(* Schneider Machine Expert - Basic project Prototype 1 Mod, file version 2.7.0.0 *)
(* ProjectInformations: Name=Nuevo proyecto *)

HARDWARE
  Cpu 0: TM221M16R/G
  ModuleExtensionObject 0: TM3DI16K
  ModuleExtensionObject 1: TM3AQ2/G
  ModuleExtensionObject 2: TM3AQ4/G
  ModuleExtensionObject 3: TM3DQ16R/G
  EthernetConfiguration: NetworkName=M221, IpAllocationMode=FixedAddress, IpAddress=0.0.0.0, SubnetMask=0.0.0.0
  SerialLineConfiguration: Baud=Baud19200, Parity=ParityEven, DataBits=DataBits8, StopBits=StopBits1, PhysicalMedium=PhysicalMediumRs485, TransmissionMode=TransmissionModeModbusRtu, SlaveId=1, Addressing=SlaveAddressing
  MastTask: UsePeriodScanMode=false, PeriodScan=100
  FastTask: Period=255
  CpuBehavior: StartingMode=StartAsPreviousState, AutoSaveRamOnEeprom=true, WatchdogPeriod=250

SYMBOLS  (address, symbol, comment, settings)
  %M0       START_BUTTON
  %M1       RESET_BUTTON
  %M2       STOP_BUTTON
  %M3       EMERGENCY_BUTTON
  %M4       AUTO_SWITCH
  %M5       ENTRY_SENSOR
  %M7       PERSON
  %M8       EXIT_SENSOR
  %M9       COUNTER_SENSOR
  %M10      ITEM_DETECTED_1
  %M11      ITEM_DETECTED_2
  %M13      MOVING_XY_1
  %M16      MOVING_Z1
  %M18      ENTRY_CONVEYOR
  %M19      MIDDLE_CONVEYOR
  %M20      EXIT_CONVEYOR
  %M21      GRAB_1
  %M22      GRAB_2
  %M23      START_LIGHT
  %M24      RESET_LIGHT
  %M25      STOP_LIGHT
  %M26      RED_LIGHT
  %M27      YELLOW_LIGHT
  %M28      GREEN_LIGHT
  %M29      ALARM
  %M100     INITIALIZE
  %M101     INITIAL_POS_1
  %M102     INITIAL_POS_2
  %M200     FLAG_AUTO
  %S21      SB_INITGRAFCET  "En el estado 1, este bit provoca una inicialización GRAFCET. Los pasos activos se desactivan y los pasos iniciales se activan"
  %X1       STATE_1
  %X2       STATE_2
  %X3       STATE_3
  %X4       STATE_4
  %X5       STATE_5
  %X6       STATE_6
  %X7       STATE_7
  %X8       STATE_8
  %X9       STATE_9
  %X10      STATE_10
  %X11      STATE_11
  %X12      STATE_12
  %X13      STATE_13
  %X14      STATE_14
  %X15      STATE_15
  %X16      STATE_16
  %X17      STATE_17
  %X18      STATE_18
  %X19      STATE_19
  %X21      STATE_21
  %MW0      X1
  %MW1      Y1
  %MW2      Z1
  %MW3      X2
  %MW4      Y2
  %MW5      Z2
  %MW6      X1_MOVE
  %MW7      Y1_MOVE
  %MW8      Z1_MOVE
  %MW9      X2_MOVE
  %MW10     Y2_MOVE
  %MW11     Z2_MOVE
  %MW12     COUNTER_OF_ITEMS
  %TM0      TIME_OF_OPERATION  [Preset=10, Base=OneSecond]
  %TM1      SECURITY_TIME  [Preset=5, Base=OneSecond]
  %TM2        "Syren time"  [Type=TOF, Preset=30, Base=OneSecond]
  %C0       NUMBER_OF_ITEMS

GRAFCET Grafcet
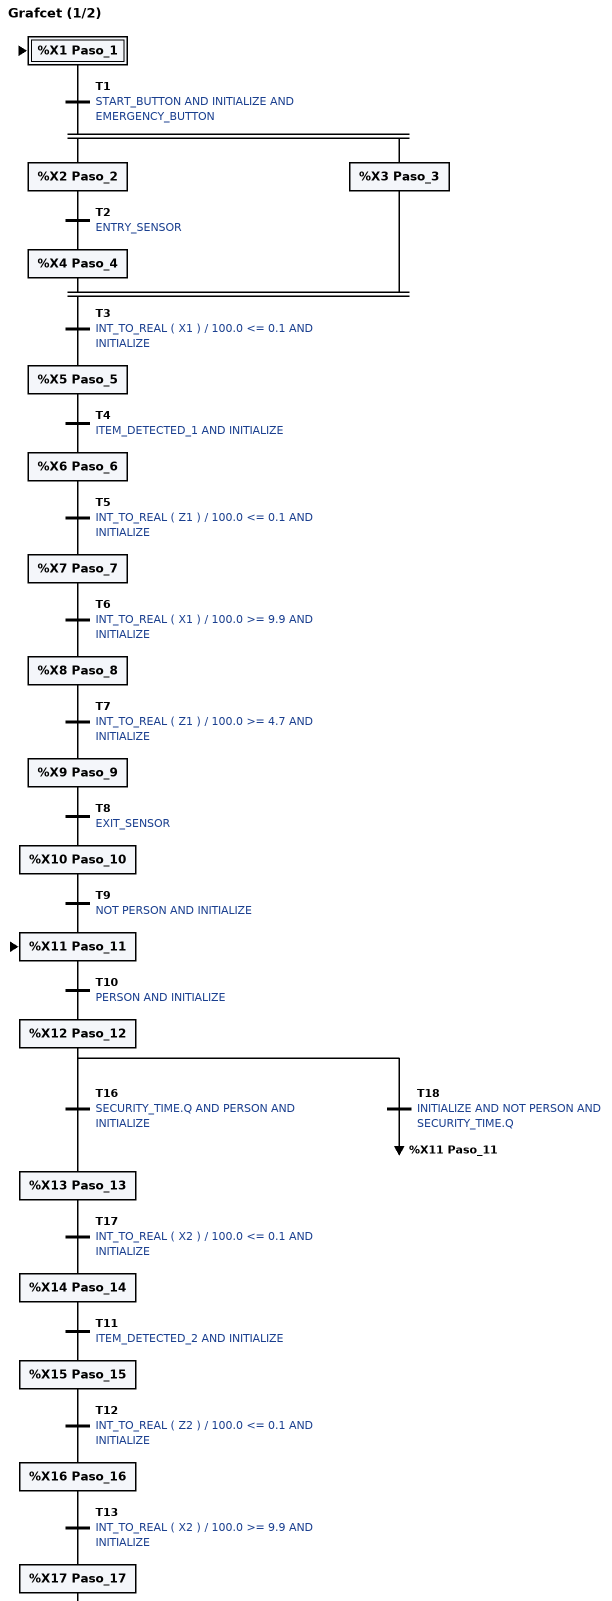
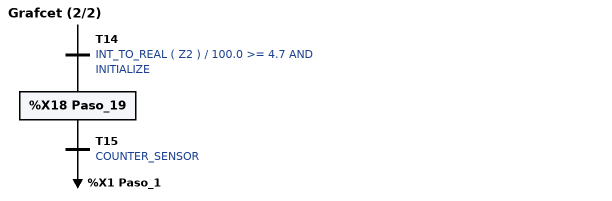
  INITIAL_STEP %X1  (* Paso_1 *)
  STEP %X2  (* Paso_2 *)
  STEP %X3  (* Paso_3 *)
  STEP %X4  (* Paso_4 *)
  STEP %X5  (* Paso_5 *)
  STEP %X6  (* Paso_6 *)
  STEP %X7  (* Paso_7 *)
  STEP %X8  (* Paso_8 *)
  STEP %X9  (* Paso_9 *)
  STEP %X10  (* Paso_10 *)
  STEP %X11  (* Paso_11 *)
  STEP %X12  (* Paso_12 *)
  STEP %X13  (* Paso_13 *)
  STEP %X14  (* Paso_14 *)
  STEP %X15  (* Paso_15 *)
  STEP %X16  (* Paso_16 *)
  STEP %X17  (* Paso_17 *)
  STEP %X18  (* Paso_19 *)
  TRANSITION T1 FROM %X1 TO %X2, %X3 := START_BUTTON AND INITIALIZE AND EMERGENCY_BUTTON;
  TRANSITION T2 FROM %X2 TO %X4 := ENTRY_SENSOR;
  TRANSITION T3 FROM %X4, %X3 TO %X5 := INT_TO_REAL ( X1 ) / 100.0 <= 0.1 AND INITIALIZE;
  TRANSITION T4 FROM %X5 TO %X6 := ITEM_DETECTED_1 AND INITIALIZE;
  TRANSITION T5 FROM %X6 TO %X7 := INT_TO_REAL ( Z1 ) / 100.0 <= 0.1 AND INITIALIZE;
  TRANSITION T6 FROM %X7 TO %X8 := INT_TO_REAL ( X1 ) / 100.0 >= 9.9 AND INITIALIZE;
  TRANSITION T7 FROM %X8 TO %X9 := INT_TO_REAL ( Z1 ) / 100.0 >= 4.7 AND INITIALIZE;
  TRANSITION T8 FROM %X9 TO %X10 := EXIT_SENSOR;
  TRANSITION T9 FROM %X10 TO %X11 := NOT PERSON AND INITIALIZE;
  TRANSITION T10 FROM %X11 TO %X12 := PERSON AND INITIALIZE;
  TRANSITION T11 FROM %X14 TO %X15 := ITEM_DETECTED_2 AND INITIALIZE;
  TRANSITION T12 FROM %X15 TO %X16 := INT_TO_REAL ( Z2 ) / 100.0 <= 0.1 AND INITIALIZE;
  TRANSITION T13 FROM %X16 TO %X17 := INT_TO_REAL ( X2 ) / 100.0 >= 9.9 AND INITIALIZE;
  TRANSITION T14 FROM %X17 TO %X18 := INT_TO_REAL ( Z2 ) / 100.0 >= 4.7 AND INITIALIZE;
  TRANSITION T15 FROM %X18 TO %X1 := COUNTER_SENSOR;
  TRANSITION T16 FROM %X12 TO %X13 := SECURITY_TIME.Q AND PERSON AND INITIALIZE;
  TRANSITION T17 FROM %X13 TO %X14 := INT_TO_REAL ( X2 ) / 100.0 <= 0.1 AND INITIALIZE;
  TRANSITION T18 FROM %X12 TO %X11 := INITIALIZE AND NOT PERSON AND SECURITY_TIME.Q;

TRANSITION T1 (%X1 -> %X2, %X3) 
  (* SectionNumber=0 *)

// Rung 0: Tr1
  LD %M0                  (* START_BUTTON *)
  AND %M100               (* INITIALIZE *)
  AND %M3                 (* EMERGENCY_BUTTON *)
  ENDT
  // as ST:
  //   TRANSITION := START_BUTTON AND INITIALIZE AND EMERGENCY_BUTTON;

TRANSITION T2 (%X2 -> %X4) 
  (* SectionNumber=0 *)

// Rung 1: Tr2
  LD %M5                  (* ENTRY_SENSOR *)
  ENDT
  // as ST:
  //   TRANSITION := ENTRY_SENSOR;

TRANSITION T3 (%X4, %X3 -> %X5) 
  (* SectionNumber=0 *)

// Rung 2: Tr3
  LD 1
  AND [ INT_TO_REAL ( %MW0 ) / 100.0 <= 0.1 ](* X1 *)
  AND %M100               (* INITIALIZE *)
  ENDT
  // as ST:
  //   TRANSITION := INT_TO_REAL ( X1 ) / 100.0 <= 0.1 AND INITIALIZE;

TRANSITION T4 (%X5 -> %X6) 
  (* SectionNumber=0 *)

// Rung 3: Tr4
  LD %M10                 (* ITEM_DETECTED_1 *)
  AND %M100               (* INITIALIZE *)
  ENDT
  // as ST:
  //   TRANSITION := ITEM_DETECTED_1 AND INITIALIZE;

TRANSITION T5 (%X6 -> %X7) 
  (* SectionNumber=0 *)

// Rung 4: Tr5
  LD 1
  AND [ INT_TO_REAL ( %MW2 ) / 100.0 <= 0.1 ](* Z1 *)
  AND %M100               (* INITIALIZE *)
  ENDT
  // as ST:
  //   TRANSITION := INT_TO_REAL ( Z1 ) / 100.0 <= 0.1 AND INITIALIZE;

TRANSITION T6 (%X7 -> %X8) 
  (* SectionNumber=0 *)

// Rung 5: Tr6
  LD 1
  AND [ INT_TO_REAL ( %MW0 ) / 100.0 >= 9.9 ](* X1 *)
  AND %M100               (* INITIALIZE *)
  ENDT
  // as ST:
  //   TRANSITION := INT_TO_REAL ( X1 ) / 100.0 >= 9.9 AND INITIALIZE;

TRANSITION T7 (%X8 -> %X9) 
  (* SectionNumber=0 *)

// Rung 6: Tr7
  LD 1
  AND [ INT_TO_REAL ( %MW2 ) / 100.0 >= 4.7 ](* Z1 *)
  AND %M100               (* INITIALIZE *)
  ENDT
  // as ST:
  //   TRANSITION := INT_TO_REAL ( Z1 ) / 100.0 >= 4.7 AND INITIALIZE;

TRANSITION T8 (%X9 -> %X10) 
  (* SectionNumber=0 *)

// Rung 7: Tr8
  LD %M8                  (* EXIT_SENSOR *)
  ENDT
  // as ST:
  //   TRANSITION := EXIT_SENSOR;

TRANSITION T9 (%X10 -> %X11) 
  (* SectionNumber=0 *)

// Rung 8: Tr9
  LDN %M7                 (* PERSON *)
  AND %M100               (* INITIALIZE *)
  ENDT
  // as ST:
  //   TRANSITION := NOT PERSON AND INITIALIZE;

TRANSITION T10 (%X11 -> %X12) 
  (* SectionNumber=0 *)

// Rung 9: Tr10
  LD %M7                  (* PERSON *)
  AND %M100               (* INITIALIZE *)
  ENDT
  // as ST:
  //   TRANSITION := PERSON AND INITIALIZE;

TRANSITION T11 (%X14 -> %X15) 
  (* SectionNumber=0 *)

// Rung 10: Tr14
  LD %M11                 (* ITEM_DETECTED_2 *)
  AND %M100               (* INITIALIZE *)
  ENDT
  // as ST:
  //   TRANSITION := ITEM_DETECTED_2 AND INITIALIZE;

TRANSITION T12 (%X15 -> %X16) 
  (* SectionNumber=0 *)

// Rung 11: Tr15
  LD 1
  AND [ INT_TO_REAL ( %MW5 ) / 100.0 <= 0.1 ](* Z2 *)
  AND %M100               (* INITIALIZE *)
  ENDT
  // as ST:
  //   TRANSITION := INT_TO_REAL ( Z2 ) / 100.0 <= 0.1 AND INITIALIZE;

TRANSITION T13 (%X16 -> %X17) 
  (* SectionNumber=0 *)

// Rung 12: Tr16
  LD 1
  AND [ INT_TO_REAL ( %MW3 ) / 100.0 >= 9.9 ](* X2 *)
  AND %M100               (* INITIALIZE *)
  ENDT
  // as ST:
  //   TRANSITION := INT_TO_REAL ( X2 ) / 100.0 >= 9.9 AND INITIALIZE;

TRANSITION T14 (%X17 -> %X18) 
  (* SectionNumber=0 *)

// Rung 13: Tr17
  LD 1
  AND [ INT_TO_REAL ( %MW5 ) / 100.0 >= 4.7 ](* Z2 *)
  AND %M100               (* INITIALIZE *)
  ENDT
  // as ST:
  //   TRANSITION := INT_TO_REAL ( Z2 ) / 100.0 >= 4.7 AND INITIALIZE;

TRANSITION T15 (%X18 -> %X1) 
  (* SectionNumber=0 *)

// Rung 14: Tr18
  LD %M9                  (* COUNTER_SENSOR *)
  ENDT
  // as ST:
  //   TRANSITION := COUNTER_SENSOR;

TRANSITION T16 (%X12 -> %X13) 
  (* SectionNumber=0 *)

// Rung 15: Tr12
  LD %TM1.Q               (* SECURITY_TIME *)
  AND %M7                 (* PERSON *)
  AND %M100               (* INITIALIZE *)
  ENDT
  // as ST:
  //   TRANSITION := SECURITY_TIME.Q AND PERSON AND INITIALIZE;

TRANSITION T17 (%X13 -> %X14) 
  (* SectionNumber=0 *)

// Rung 16: Tr13
  LD 1
  AND [ INT_TO_REAL ( %MW3 ) / 100.0 <= 0.1 ](* X2 *)
  AND %M100               (* INITIALIZE *)
  ENDT
  // as ST:
  //   TRANSITION := INT_TO_REAL ( X2 ) / 100.0 <= 0.1 AND INITIALIZE;

TRANSITION T18 (%X12 -> %X11) 
  (* SectionNumber=0 *)

// Rung 17: Tr11
  LD %M100                (* INITIALIZE *)
  ANDN %M7                (* PERSON *)
  AND %TM1.Q              (* SECURITY_TIME *)
  ENDT
  // as ST:
  //   TRANSITION := INITIALIZE AND NOT PERSON AND SECURITY_TIME.Q;

POU Actions
  (* SectionNumber=20 *)

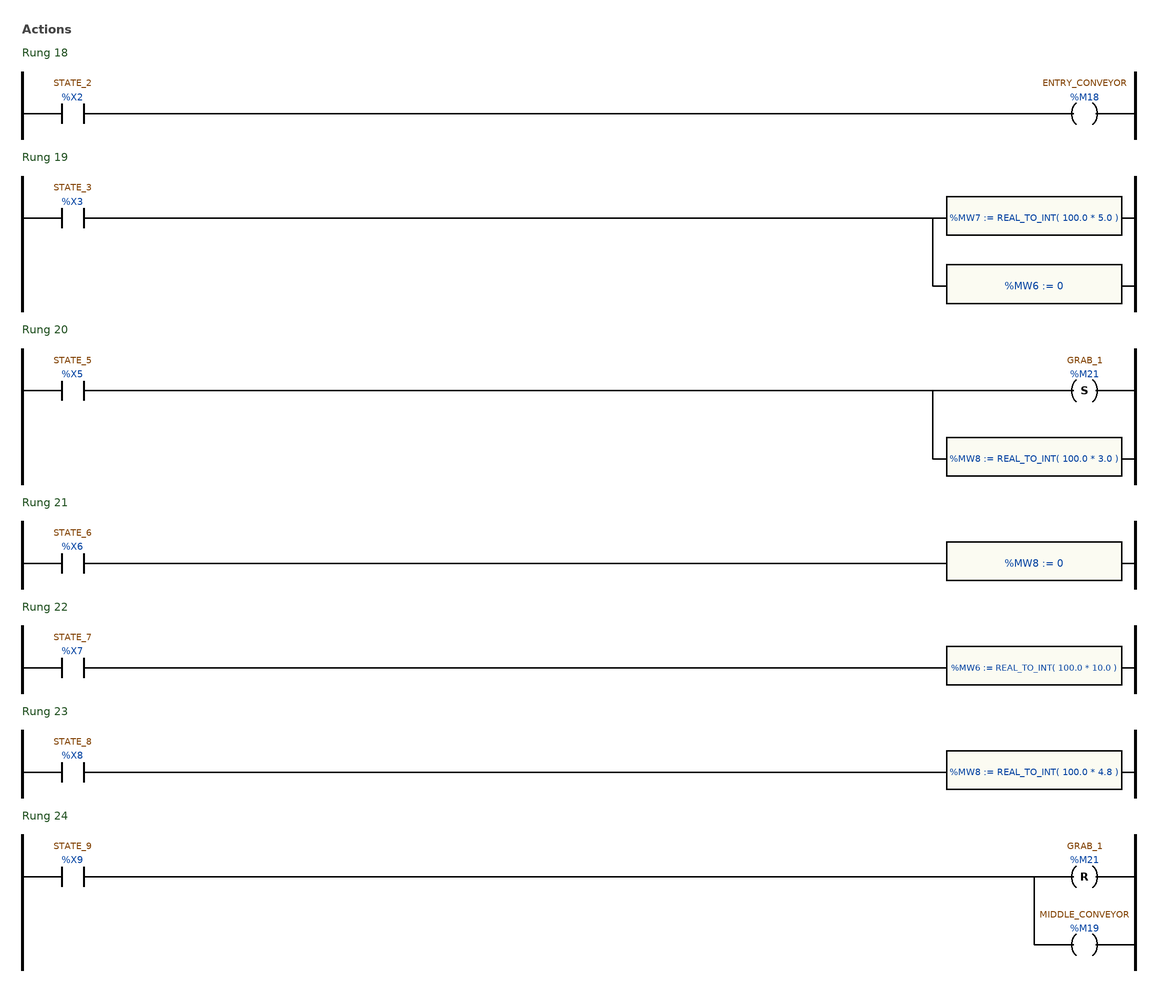

// Rung 18
  LD %X2                  (* STATE_2 *)
  ST %M18                 (* ENTRY_CONVEYOR *)
  // as ST:
  //   ENTRY_CONVEYOR := STATE_2;

// Rung 19
  LD %X3                  (* STATE_3 *)
  [ %MW7 := REAL_TO_INT ( 100.0 * 5.0 ) ](* Y1_MOVE *)
  [ %MW6 := 0 ]           (* X1_MOVE *)
  // as ST:
  //   IF STATE_3 THEN Y1_MOVE := REAL_TO_INT ( 100.0 * 5.0 ); END_IF;
  //   IF STATE_3 THEN X1_MOVE := 0; END_IF;

// Rung 20
  LD %X5                  (* STATE_5 *)
  S %M21                  (* GRAB_1 *)
  [ %MW8 := REAL_TO_INT ( 100.0 * 3.0 ) ](* Z1_MOVE *)
  // as ST:
  //   IF STATE_5 THEN GRAB_1 := TRUE; END_IF;
  //   IF STATE_5 THEN Z1_MOVE := REAL_TO_INT ( 100.0 * 3.0 ); END_IF;

// Rung 21
  LD %X6                  (* STATE_6 *)
  [ %MW8 := 0 ]           (* Z1_MOVE *)
  // as ST:
  //   IF STATE_6 THEN Z1_MOVE := 0; END_IF;

// Rung 22
  LD %X7                  (* STATE_7 *)
  [ %MW6 := REAL_TO_INT ( 100.0 * 10.0 ) ](* X1_MOVE *)
  // as ST:
  //   IF STATE_7 THEN X1_MOVE := REAL_TO_INT ( 100.0 * 10.0 ); END_IF;

// Rung 23
  LD %X8                  (* STATE_8 *)
  [ %MW8 := REAL_TO_INT ( 100.0 * 4.8 ) ](* Z1_MOVE *)
  // as ST:
  //   IF STATE_8 THEN Z1_MOVE := REAL_TO_INT ( 100.0 * 4.8 ); END_IF;

// Rung 24
  LD %X9                  (* STATE_9 *)
  R %M21                  (* GRAB_1 *)
  ST %M19                 (* MIDDLE_CONVEYOR *)
  // as ST:
  //   IF STATE_9 THEN GRAB_1 := FALSE; END_IF;
  //   MIDDLE_CONVEYOR := STATE_9;

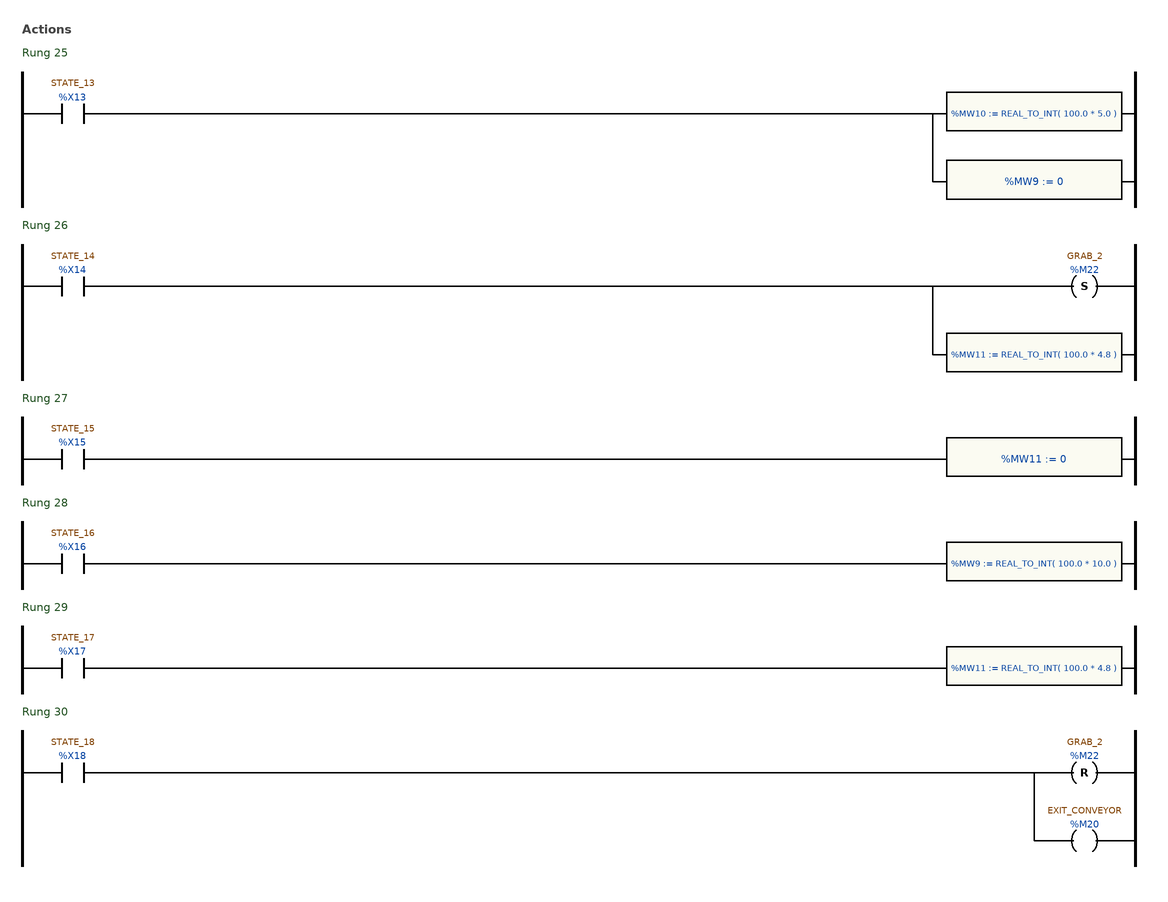

// Rung 25
  LD %X13                 (* STATE_13 *)
  [ %MW10 := REAL_TO_INT ( 100.0 * 5.0 ) ](* Y2_MOVE *)
  [ %MW9 := 0 ]           (* X2_MOVE *)
  // as ST:
  //   IF STATE_13 THEN Y2_MOVE := REAL_TO_INT ( 100.0 * 5.0 ); END_IF;
  //   IF STATE_13 THEN X2_MOVE := 0; END_IF;

// Rung 26
  LD %X14                 (* STATE_14 *)
  S %M22                  (* GRAB_2 *)
  [ %MW11 := REAL_TO_INT ( 100.0 * 4.8 ) ](* Z2_MOVE *)
  // as ST:
  //   IF STATE_14 THEN GRAB_2 := TRUE; END_IF;
  //   IF STATE_14 THEN Z2_MOVE := REAL_TO_INT ( 100.0 * 4.8 ); END_IF;

// Rung 27
  LD %X15                 (* STATE_15 *)
  [ %MW11 := 0 ]          (* Z2_MOVE *)
  // as ST:
  //   IF STATE_15 THEN Z2_MOVE := 0; END_IF;

// Rung 28
  LD %X16                 (* STATE_16 *)
  [ %MW9 := REAL_TO_INT ( 100.0 * 10.0 ) ](* X2_MOVE *)
  // as ST:
  //   IF STATE_16 THEN X2_MOVE := REAL_TO_INT ( 100.0 * 10.0 ); END_IF;

// Rung 29
  LD %X17                 (* STATE_17 *)
  [ %MW11 := REAL_TO_INT ( 100.0 * 4.8 ) ](* Z2_MOVE *)
  // as ST:
  //   IF STATE_17 THEN Z2_MOVE := REAL_TO_INT ( 100.0 * 4.8 ); END_IF;

// Rung 30
  LD %X18                 (* STATE_18 *)
  R %M22                  (* GRAB_2 *)
  ST %M20                 (* EXIT_CONVEYOR *)
  // as ST:
  //   IF STATE_18 THEN GRAB_2 := FALSE; END_IF;
  //   EXIT_CONVEYOR := STATE_18;

POU Buttons
  (* SectionNumber=21 *)

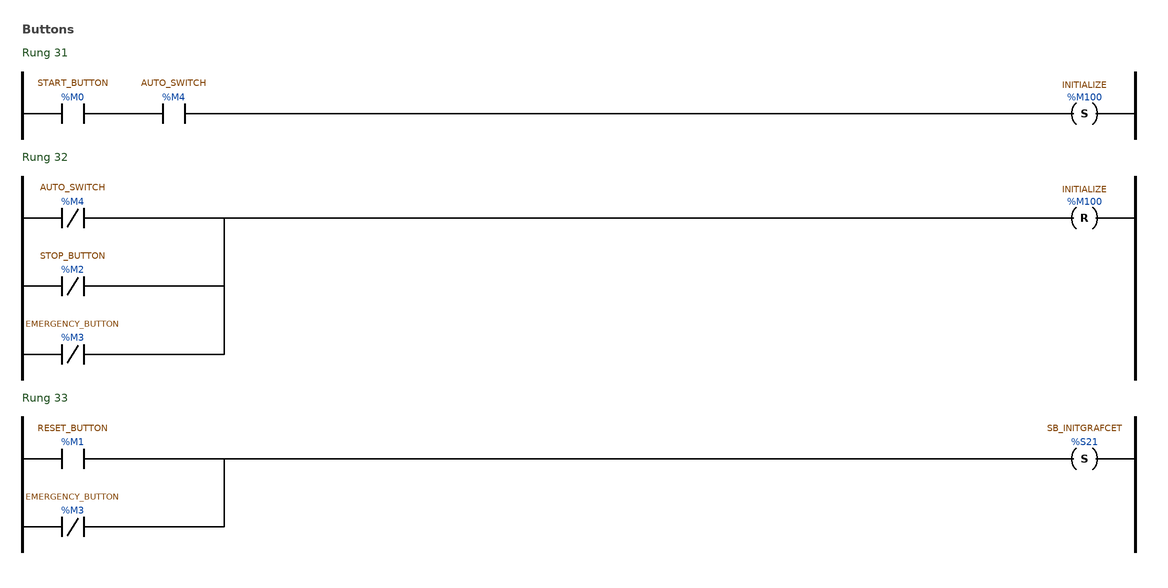

// Rung 31
  LD %M0                  (* START_BUTTON *)
  AND %M4                 (* AUTO_SWITCH *)
  S %M100                 (* INITIALIZE *)
  // as ST:
  //   IF START_BUTTON AND AUTO_SWITCH THEN INITIALIZE := TRUE; END_IF;

// Rung 32
  LDN %M4                 (* AUTO_SWITCH *)
  ORN %M2                 (* STOP_BUTTON *)
  ORN %M3                 (* EMERGENCY_BUTTON *)
  R %M100                 (* INITIALIZE *)
  // as ST:
  //   IF NOT AUTO_SWITCH OR NOT STOP_BUTTON OR NOT EMERGENCY_BUTTON THEN INITIALIZE := FALSE; END_IF;

// Rung 33
  LD %M1                  (* RESET_BUTTON *)
  ORN %M3                 (* EMERGENCY_BUTTON *)
  S %S21                  (* SB_INITGRAFCET *)
  // as ST:
  //   IF RESET_BUTTON OR NOT EMERGENCY_BUTTON THEN SB_INITGRAFCET := TRUE; END_IF;

POU Timers and Counters
  (* SectionNumber=22 *)

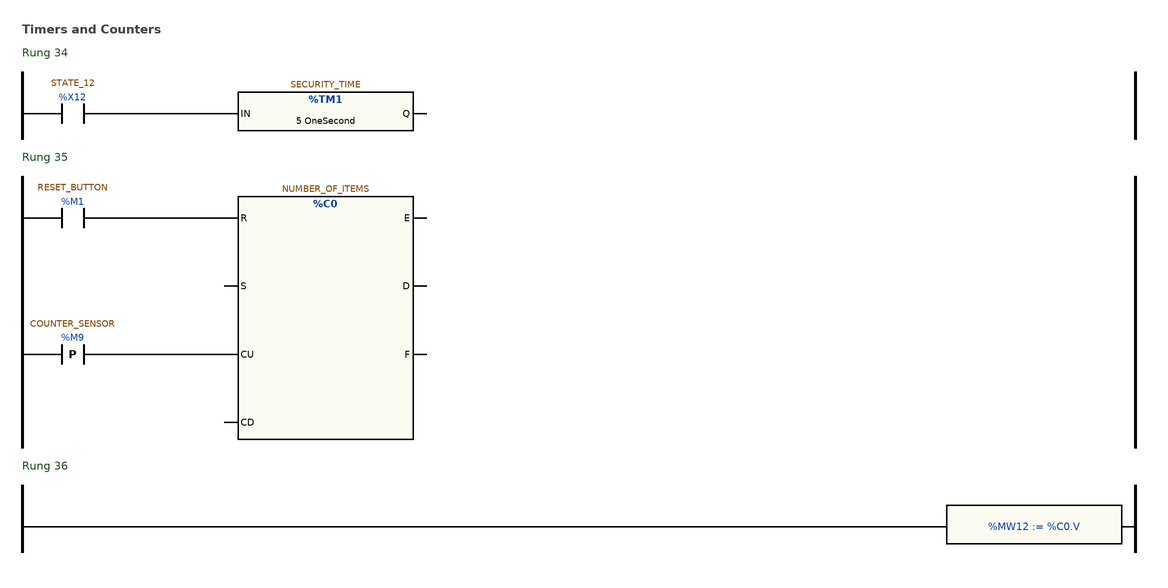

// Rung 34
  BLK %TM1                (* SECURITY_TIME *)
  LD %X12                 (* STATE_12 *)
  IN
  END_BLK
  // as ST:
  //   SECURITY_TIME(IN := STATE_12);

// Rung 35
  BLK %C0                 (* NUMBER_OF_ITEMS *)
  LD %M1                  (* RESET_BUTTON *)
  R
  LDR %M9                 (* COUNTER_SENSOR *)
  CU
  END_BLK
  // as ST:
  //   NUMBER_OF_ITEMS(R := RESET_BUTTON, CU := RISING(COUNTER_SENSOR));

// Rung 36
  LD 1
  [ %MW12 := %C0.V ]      (* COUNTER_OF_ITEMS, NUMBER_OF_ITEMS *)
  // as ST:
  //   COUNTER_OF_ITEMS := NUMBER_OF_ITEMS.V;

POU Initial conditions
  (* SectionNumber=23 *)

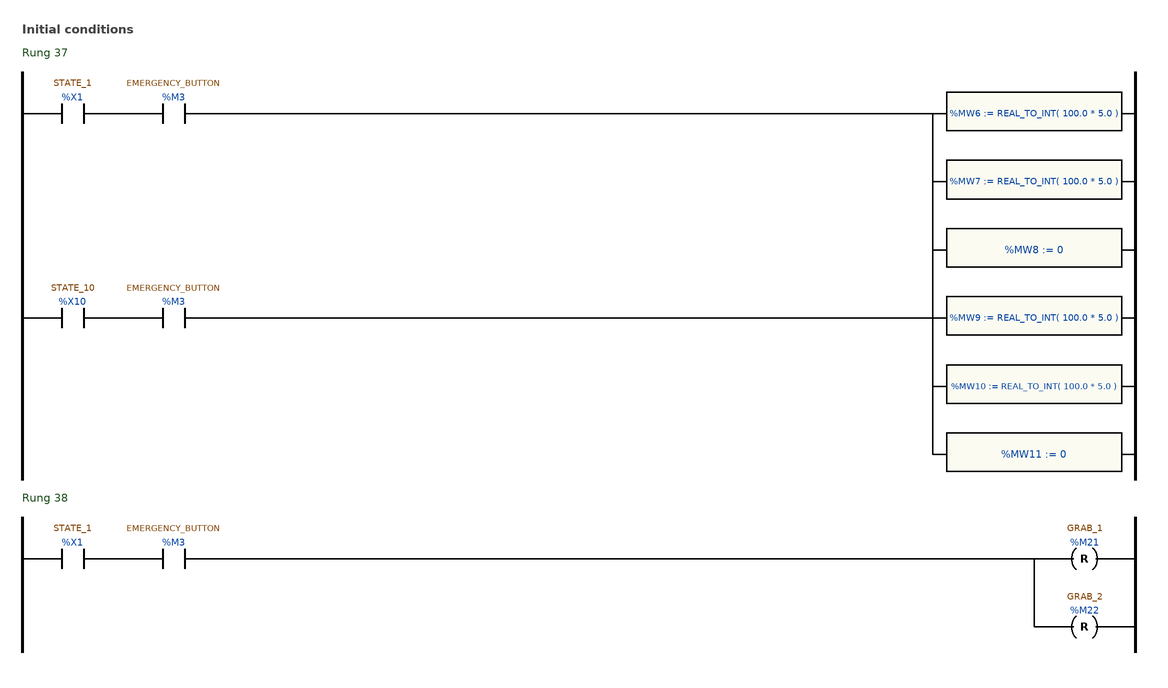

// Rung 37
  LD %X1                  (* STATE_1 *)
  AND %M3                 (* EMERGENCY_BUTTON *)
  OR( %X10                (* STATE_10 *)
  AND %M3                 (* EMERGENCY_BUTTON *)
  )
  [ %MW6 := REAL_TO_INT ( 100.0 * 5.0 ) ](* X1_MOVE *)
  [ %MW7 := REAL_TO_INT ( 100.0 * 5.0 ) ](* Y1_MOVE *)
  [ %MW8 := 0 ]           (* Z1_MOVE *)
  [ %MW9 := REAL_TO_INT ( 100.0 * 5.0 ) ](* X2_MOVE *)
  [ %MW10 := REAL_TO_INT ( 100.0 * 5.0 ) ](* Y2_MOVE *)
  [ %MW11 := 0 ]          (* Z2_MOVE *)
  // as ST:
  //   IF STATE_1 AND EMERGENCY_BUTTON OR STATE_10 AND EMERGENCY_BUTTON THEN X1_MOVE := REAL_TO_INT ( 100.0 * 5.0 ); END_IF;
  //   IF STATE_1 AND EMERGENCY_BUTTON OR STATE_10 AND EMERGENCY_BUTTON THEN Y1_MOVE := REAL_TO_INT ( 100.0 * 5.0 ); END_IF;
  //   IF STATE_1 AND EMERGENCY_BUTTON OR STATE_10 AND EMERGENCY_BUTTON THEN Z1_MOVE := 0; END_IF;
  //   IF STATE_1 AND EMERGENCY_BUTTON OR STATE_10 AND EMERGENCY_BUTTON THEN X2_MOVE := REAL_TO_INT ( 100.0 * 5.0 ); END_IF;
  //   IF STATE_1 AND EMERGENCY_BUTTON OR STATE_10 AND EMERGENCY_BUTTON THEN Y2_MOVE := REAL_TO_INT ( 100.0 * 5.0 ); END_IF;
  //   IF STATE_1 AND EMERGENCY_BUTTON OR STATE_10 AND EMERGENCY_BUTTON THEN Z2_MOVE := 0; END_IF;

// Rung 38
  LD %X1                  (* STATE_1 *)
  AND %M3                 (* EMERGENCY_BUTTON *)
  R %M21                  (* GRAB_1 *)
  R %M22                  (* GRAB_2 *)
  // as ST:
  //   IF STATE_1 AND EMERGENCY_BUTTON THEN GRAB_1 := FALSE; END_IF;
  //   IF STATE_1 AND EMERGENCY_BUTTON THEN GRAB_2 := FALSE; END_IF;

POU Lights and warnings
  (* SectionNumber=24 *)

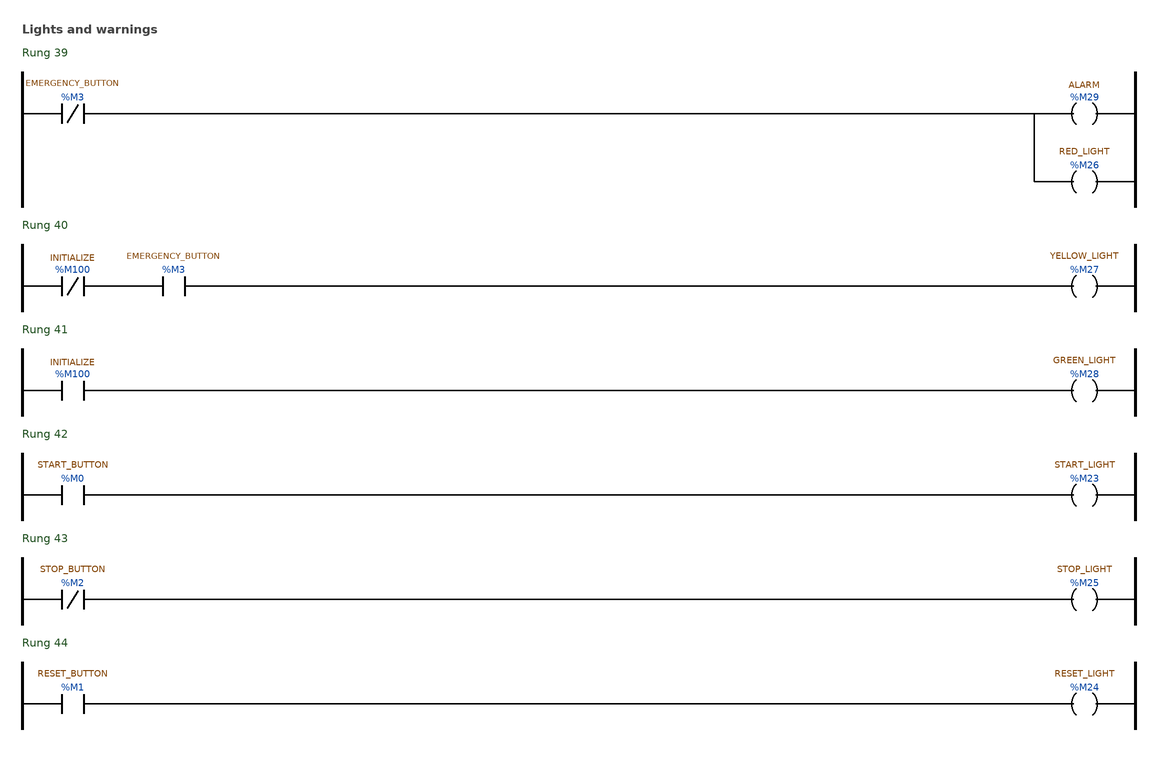

// Rung 39
  LDN %M3                 (* EMERGENCY_BUTTON *)
  ST %M29                 (* ALARM *)
  ST %M26                 (* RED_LIGHT *)
  // as ST:
  //   ALARM := NOT EMERGENCY_BUTTON;
  //   RED_LIGHT := NOT EMERGENCY_BUTTON;

// Rung 40
  LDN %M100               (* INITIALIZE *)
  AND %M3                 (* EMERGENCY_BUTTON *)
  ST %M27                 (* YELLOW_LIGHT *)
  // as ST:
  //   YELLOW_LIGHT := NOT INITIALIZE AND EMERGENCY_BUTTON;

// Rung 41
  LD %M100                (* INITIALIZE *)
  ST %M28                 (* GREEN_LIGHT *)
  // as ST:
  //   GREEN_LIGHT := INITIALIZE;

// Rung 42
  LD %M0                  (* START_BUTTON *)
  ST %M23                 (* START_LIGHT *)
  // as ST:
  //   START_LIGHT := START_BUTTON;

// Rung 43
  LDN %M2                 (* STOP_BUTTON *)
  ST %M25                 (* STOP_LIGHT *)
  // as ST:
  //   STOP_LIGHT := NOT STOP_BUTTON;

// Rung 44
  LD %M1                  (* RESET_BUTTON *)
  ST %M24                 (* RESET_LIGHT *)
  // as ST:
  //   RESET_LIGHT := RESET_BUTTON;
